VAR_GLOBAL
    g_aSensorBuffer : ARRAY[0..g_aSensorBuffers, 0..g_aSensorBufferSize] OF ST_SensorData; // aSensorBuffers buffers of aSensorBufferSize samples each
    g_aWriteSQL     : ARRAY[0..g_ASensorBuffers] OF BOOL;                 // Marks buffers ready for DB insert
	
END_VAR

VAR_GLOBAL CONSTANT
	g_aSensorBufferSize : INT := 999;
	g_aSensorBuffers : INT := 100;
	sLocalID : STRING := '145.44.56.240.1.1'; //ams net id of database host
END_VAR

(* stored: Version 1.1.0.1
   GVL Global_Variables: Id {592dda55-669d-4363-87cb-faf5f8692ce1} *)
